// TIA Portal V17 export
// export: Created 2023-04-04T07:17:21.5901829Z, ExportSetting WithDefaults, DisplayName Totally Integrated Automation Portal, DisplayVersion V17 Update 4, DisplayName TIA Portal Openness, DisplayVersion V17 Update 4, DisplayName TIA Portal Version Control Interface, DisplayVersion V17, DisplayName STEP 7 Professional, DisplayVersion V17 Update 4, DisplayName STEP 7 Safety, DisplayVersion V17, DisplayName WinCC Professional, DisplayVersion V17 Update 4
FUNCTION "MV SKID (PE)_1" : Void   // FC45, LAD
TITLE = ModBus TCP for MVSKID Power Electronics
{ S7_Optimized_Access := 'TRUE' }
VERSION : 0.1
// stored: AutoNumber false, IsIECCheckEnabled false, SetENOAutomatically false, UDAEnableTagReadback false
   VAR_TEMP   // added for the SCL form of the ladder/FBD networks
      _w1 : Bool;
   END_VAR
BEGIN

REGION Network 1: Function Modbus Client
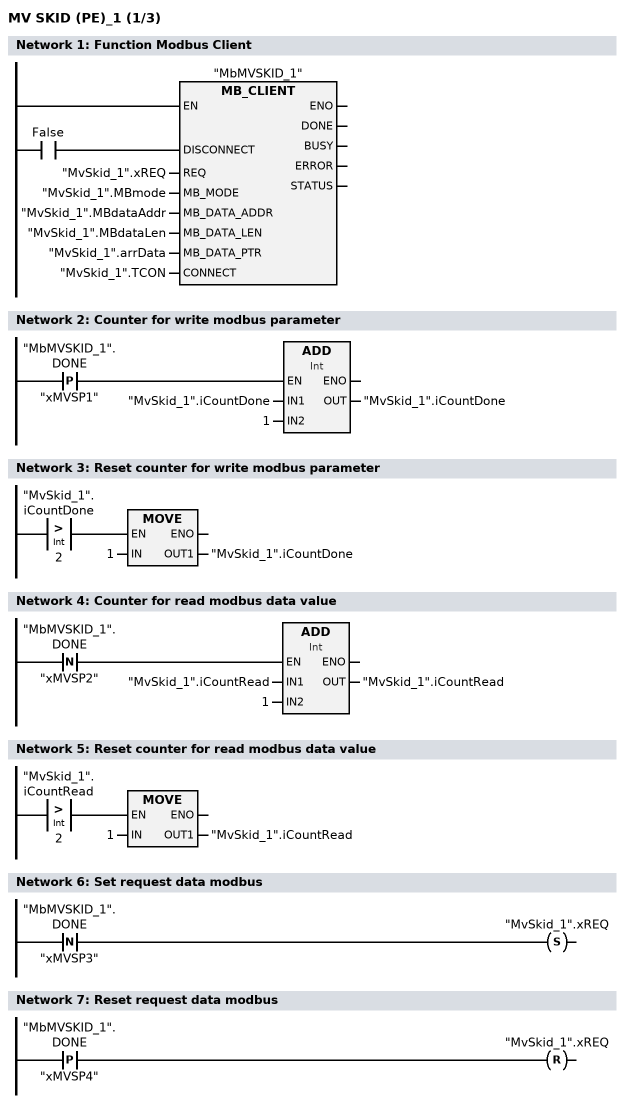
   RUNG wire#powerrail
      "MbMVSKID_1".MB_CLIENT(DISCONNECT := wire#w1, REQ := "MvSkid_1".xREQ, MB_MODE := "MvSkid_1".MBmode, MB_DATA_ADDR := "MvSkid_1".MBdataAddr, MB_DATA_LEN := "MvSkid_1".MBdataLen, MB_DATA_PTR := "MvSkid_1".arrData, CONNECT := "MvSkid_1".TCON, DONE =>, BUSY =>, ERROR =>, STATUS =>)
   END_RUNG
   RUNG wire#powerrail
      Contact( False )
   END_RUNG wire#w1
   // the same network as SCL:
   "MbMVSKID_1"(DISCONNECT := False,   // MB_CLIENT
                REQ := "MvSkid_1".xREQ,
                MB_MODE := "MvSkid_1".MBmode,
                MB_DATA_ADDR := "MvSkid_1".MBdataAddr,
                MB_DATA_LEN := "MvSkid_1".MBdataLen,
                MB_DATA_PTR := "MvSkid_1".arrData,
                CONNECT := "MvSkid_1".TCON);
END_REGION

REGION Network 2: Counter for write modbus parameter
   RUNG wire#powerrail
      P_Contact(operand := "MbMVSKID_1".DONE, bit := "xMVSP1")
      { S7_Templates := "SrcType := Int" } Add(in1 := "MvSkid_1".iCountDone, in2 := 1, out => "MvSkid_1".iCountDone)
   END_RUNG
   // the same network as SCL:
   #_w1 := "MbMVSKID_1".DONE AND NOT "xMVSP1";   // rising edge of "MbMVSKID_1".DONE
   "xMVSP1" := "MbMVSKID_1".DONE;
   IF #_w1 THEN "MvSkid_1".iCountDone := "MvSkid_1".iCountDone + 1; END_IF;
END_REGION

REGION Network 3: Reset counter for write modbus parameter
   RUNG wire#powerrail
      { S7_Templates := "SrcType := Int" } GT_Contact(in1 := "MvSkid_1".iCountDone, in2 := 2)
      Move(in := 1, out1 => "MvSkid_1".iCountDone)
   END_RUNG
   // the same network as SCL:
   IF "MvSkid_1".iCountDone > 2 THEN "MvSkid_1".iCountDone := 1; END_IF;
END_REGION

REGION Network 4: Counter for read modbus data value
   RUNG wire#powerrail
      N_Contact(operand := "MbMVSKID_1".DONE, bit := "xMVSP2")
      { S7_Templates := "SrcType := Int" } Add(in1 := "MvSkid_1".iCountRead, in2 := 1, out => "MvSkid_1".iCountRead)
   END_RUNG
   // the same network as SCL:
   #_w1 := NOT "MbMVSKID_1".DONE AND "xMVSP2";   // falling edge of "MbMVSKID_1".DONE
   "xMVSP2" := "MbMVSKID_1".DONE;
   IF #_w1 THEN "MvSkid_1".iCountRead := "MvSkid_1".iCountRead + 1; END_IF;
END_REGION

REGION Network 5: Reset counter for read modbus data value
   RUNG wire#powerrail
      { S7_Templates := "SrcType := Int" } GT_Contact(in1 := "MvSkid_1".iCountRead, in2 := 2)
      Move(in := 1, out1 => "MvSkid_1".iCountRead)
   END_RUNG
   // the same network as SCL:
   IF "MvSkid_1".iCountRead > 2 THEN "MvSkid_1".iCountRead := 1; END_IF;
END_REGION

REGION Network 6: Set request data modbus
   RUNG wire#powerrail
      N_Contact(operand := "MbMVSKID_1".DONE, bit := "xMVSP3")
      S_Coil( "MvSkid_1".xREQ )
   END_RUNG
   // the same network as SCL:
   #_w1 := NOT "MbMVSKID_1".DONE AND "xMVSP3";   // falling edge of "MbMVSKID_1".DONE
   "xMVSP3" := "MbMVSKID_1".DONE;
   IF #_w1 THEN "MvSkid_1".xREQ := TRUE; END_IF;
END_REGION

REGION Network 7: Reset request data modbus
   RUNG wire#powerrail
      P_Contact(operand := "MbMVSKID_1".DONE, bit := "xMVSP4")
      R_Coil( "MvSkid_1".xREQ )
   END_RUNG
   // the same network as SCL:
   #_w1 := "MbMVSKID_1".DONE AND NOT "xMVSP4";   // rising edge of "MbMVSKID_1".DONE
   "xMVSP4" := "MbMVSKID_1".DONE;
   IF #_w1 THEN "MvSkid_1".xREQ := FALSE; END_IF;
END_REGION

REGION Network 8: Write R_MVSKID parameter
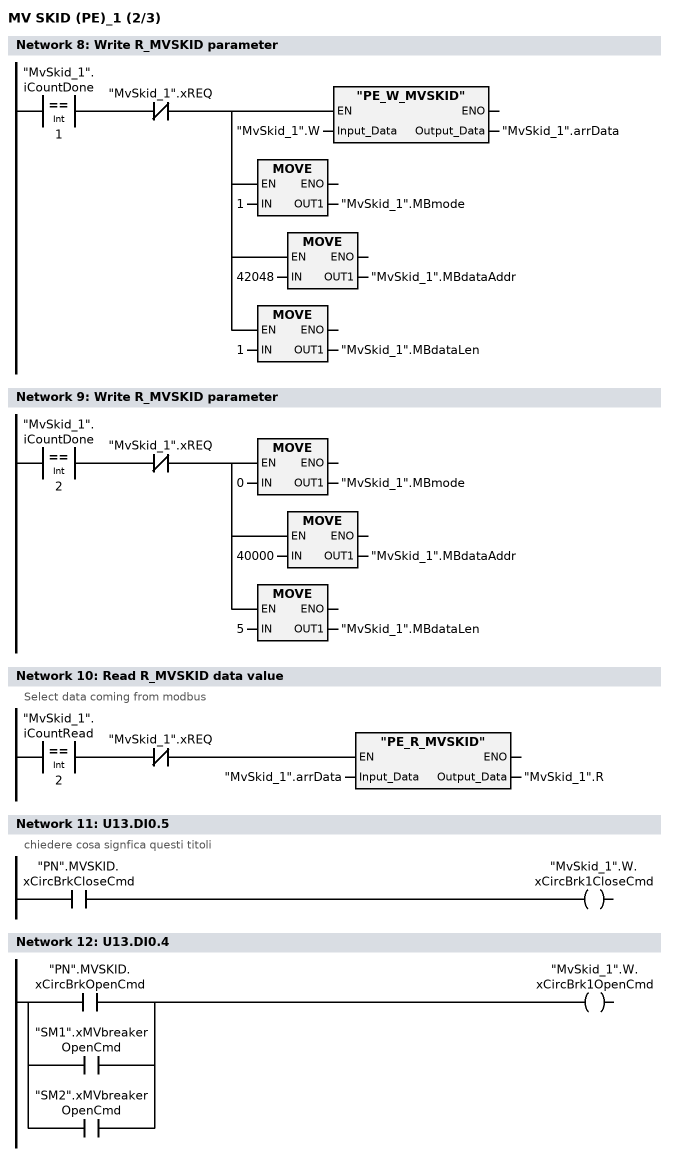
   RUNG wire#powerrail
      { S7_Templates := "SrcType := Int" } EQ_Contact(in1 := "MvSkid_1".iCountDone, in2 := 1)
      I_Contact( "MvSkid_1".xREQ )
      wire#w1
      "PE_W_MVSKID"(Input_Data := "MvSkid_1".W, Output_Data => "MvSkid_1".arrData)
   END_RUNG
   RUNG wire#w1
      Move(in := 1, out1 => "MvSkid_1".MBmode)
   END_RUNG
   RUNG wire#w1
      Move(in := 42048, out1 => "MvSkid_1".MBdataAddr)
   END_RUNG
   RUNG wire#w1
      Move(in := 1, out1 => "MvSkid_1".MBdataLen)
   END_RUNG
   // the same network as SCL:
   #_w1 := ("MvSkid_1".iCountDone = 1) AND NOT "MvSkid_1".xREQ;
   IF #_w1 THEN
       "PE_W_MVSKID"(Input_Data := "MvSkid_1".W, Output_Data => "MvSkid_1".arrData);
       "MvSkid_1".MBmode := 1;
       "MvSkid_1".MBdataAddr := 42048;
       "MvSkid_1".MBdataLen := 1;
   END_IF;
END_REGION

REGION Network 9: Write R_MVSKID parameter
   RUNG wire#powerrail
      { S7_Templates := "SrcType := Int" } EQ_Contact(in1 := "MvSkid_1".iCountDone, in2 := 2)
      I_Contact( "MvSkid_1".xREQ )
      wire#w1
      Move(in := 0, out1 => "MvSkid_1".MBmode)
   END_RUNG
   RUNG wire#w1
      Move(in := 40000, out1 => "MvSkid_1".MBdataAddr)
   END_RUNG
   RUNG wire#w1
      Move(in := 5, out1 => "MvSkid_1".MBdataLen)
   END_RUNG
   // the same network as SCL:
   IF ("MvSkid_1".iCountDone = 2) AND NOT "MvSkid_1".xREQ THEN
       "MvSkid_1".MBmode := 0;
       "MvSkid_1".MBdataAddr := 40000;
       "MvSkid_1".MBdataLen := 5;
   END_IF;
END_REGION

REGION Network 10: Read R_MVSKID data value
   // Select data coming from modbus
   RUNG wire#powerrail
      { S7_Templates := "SrcType := Int" } EQ_Contact(in1 := "MvSkid_1".iCountRead, in2 := 2)
      I_Contact( "MvSkid_1".xREQ )
      "PE_R_MVSKID"(Input_Data := "MvSkid_1".arrData, Output_Data => "MvSkid_1".R)
   END_RUNG
   // the same network as SCL:
   IF ("MvSkid_1".iCountRead = 2) AND NOT "MvSkid_1".xREQ THEN
       "PE_R_MVSKID"(Input_Data := "MvSkid_1".arrData, Output_Data => "MvSkid_1".R);
   END_IF;
END_REGION

REGION Network 11: U13.DI0.5
   // chiedere cosa signfica questi titoli
   RUNG wire#powerrail
      Contact( "PN".MVSKID.xCircBrkCloseCmd )
      Coil( "MvSkid_1".W.xCircBrk1CloseCmd )
   END_RUNG
   // the same network as SCL:
   "MvSkid_1".W.xCircBrk1CloseCmd := "PN".MVSKID.xCircBrkCloseCmd;
END_REGION

REGION Network 12: U13.DI0.4
   RUNG wire#powerrail
      Contact( "PN".MVSKID.xCircBrkOpenCmd )
      wire#w1
      Coil( "MvSkid_1".W.xCircBrk1OpenCmd )
   END_RUNG
   RUNG wire#powerrail
      Contact( "SM1".xMVbreakerOpenCmd )
   END_RUNG wire#w1
   RUNG wire#powerrail
      Contact( "SM2".xMVbreakerOpenCmd )
   END_RUNG wire#w1
   // the same network as SCL:
   "MvSkid_1".W.xCircBrk1OpenCmd := "PN".MVSKID.xCircBrkOpenCmd OR "SM1".xMVbreakerOpenCmd OR "SM2".xMVbreakerOpenCmd;
END_REGION

REGION Network 13: MV SKID Fault
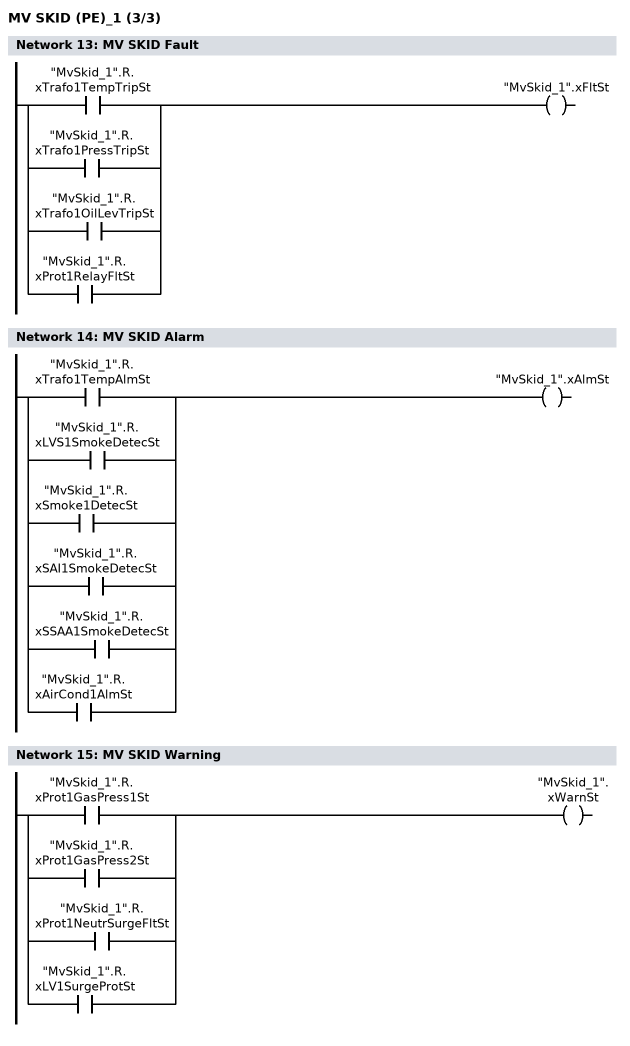
   RUNG wire#powerrail
      Contact( "MvSkid_1".R.xTrafo1TempTripSt )
      wire#w1
      Coil( "MvSkid_1".xFltSt )
   END_RUNG
   RUNG wire#powerrail
      Contact( "MvSkid_1".R.xTrafo1PressTripSt )
   END_RUNG wire#w1
   RUNG wire#powerrail
      Contact( "MvSkid_1".R.xTrafo1OilLevTripSt )
   END_RUNG wire#w1
   RUNG wire#powerrail
      Contact( "MvSkid_1".R.xProt1RelayFltSt )
   END_RUNG wire#w1
   // the same network as SCL:
   "MvSkid_1".xFltSt := "MvSkid_1".R.xTrafo1TempTripSt OR "MvSkid_1".R.xTrafo1PressTripSt OR "MvSkid_1".R.xTrafo1OilLevTripSt OR "MvSkid_1".R.xProt1RelayFltSt;
END_REGION

REGION Network 14: MV SKID Alarm
   RUNG wire#powerrail
      Contact( "MvSkid_1".R.xTrafo1TempAlmSt )
      wire#w1
      Coil( "MvSkid_1".xAlmSt )
   END_RUNG
   RUNG wire#powerrail
      Contact( "MvSkid_1".R.xLVS1SmokeDetecSt )
   END_RUNG wire#w1
   RUNG wire#powerrail
      Contact( "MvSkid_1".R.xSmoke1DetecSt )
   END_RUNG wire#w1
   RUNG wire#powerrail
      Contact( "MvSkid_1".R.xSAI1SmokeDetecSt )
   END_RUNG wire#w1
   RUNG wire#powerrail
      Contact( "MvSkid_1".R.xSSAA1SmokeDetecSt )
   END_RUNG wire#w1
   RUNG wire#powerrail
      Contact( "MvSkid_1".R.xAirCond1AlmSt )
   END_RUNG wire#w1
   // the same network as SCL:
   "MvSkid_1".xAlmSt := "MvSkid_1".R.xTrafo1TempAlmSt OR "MvSkid_1".R.xLVS1SmokeDetecSt OR "MvSkid_1".R.xSmoke1DetecSt OR "MvSkid_1".R.xSAI1SmokeDetecSt OR "MvSkid_1".R.xSSAA1SmokeDetecSt OR "MvSkid_1".R.xAirCond1AlmSt;
END_REGION

REGION Network 15: MV SKID Warning
   RUNG wire#powerrail
      Contact( "MvSkid_1".R.xProt1GasPress1St )
      wire#w1
      Coil( "MvSkid_1".xWarnSt )
   END_RUNG
   RUNG wire#powerrail
      Contact( "MvSkid_1".R.xProt1GasPress2St )
   END_RUNG wire#w1
   RUNG wire#powerrail
      Contact( "MvSkid_1".R.xProt1NeutrSurgeFltSt )
   END_RUNG wire#w1
   RUNG wire#powerrail
      Contact( "MvSkid_1".R.xLV1SurgeProtSt )
   END_RUNG wire#w1
   // the same network as SCL:
   "MvSkid_1".xWarnSt := "MvSkid_1".R.xProt1GasPress1St OR "MvSkid_1".R.xProt1GasPress2St OR "MvSkid_1".R.xProt1NeutrSurgeFltSt OR "MvSkid_1".R.xLV1SurgeProtSt;
END_REGION

REGION Network 16 (SCL): MV SKID Line Disconnector & Breaker Status
   "MvSkid_1".wLine1DiscSt.%X0 := "MvSkid_1".R.xLine1DiscOpenSt;
   "MvSkid_1".wLine1DiscSt.%X1 := "MvSkid_1".R.xLine1DiscCloseSt;
   "MvSkid_1".wLine1DiscSt.%X2 := "MvSkid_1".R.xLine1GndCloseSt;

   "MvSkid_1".wLine2DiscSt.%X0 := "MvSkid_1".R.xLine2DiscOpenSt;
   "MvSkid_1".wLine2DiscSt.%X1 := "MvSkid_1".R.xLine2DiscCloseSt;
   "MvSkid_1".wLine2DiscSt.%X2 := "MvSkid_1".R.xLine2GndCloseSt;

   "MvSkid_1".wProt1DiscSt.%X0 := "MvSkid_1".R.xProt1DiscOpenSt;
   "MvSkid_1".wProt1DiscSt.%X1 := "MvSkid_1".R.xProt1DiscCloseSt;
   "MvSkid_1".wProt1DiscSt.%X2 := "MvSkid_1".R.xProt1GndCloseSt;

   "MvSkid_1".wProt1CircBrkSt.%X0 := "MvSkid_1".R.xProt1CircBrkOpenSt;
   "MvSkid_1".wProt1CircBrkSt.%X1 := "MvSkid_1".R.xProt1CircBrkCloseSt;
END_REGION
END_FUNCTION
